{attribute 'qualified_only'}
VAR_GLOBAL
	Switch:BOOL;
	Lamp:bool;
END_VAR

(* stored: Version 1.1.0.1, ProductVersion 3.1.4024.5
   GVL GVL1: Id {4139258c-4b3d-4129-8a85-55cda263a2ff} *)
